PROGRAM sub_Light
VAR
		fbLichtHausgang 		: FB_Light;
		fbLichtTechnikraum 		: FB_Light;
		fbLichtHobbyraum 		: FB_Light;
		fbLichtKueche			: FB_Light;
		fbLichtWerkstatt		: FB_Light;
		fbLichtGarage			: FB_Light;
		fbLichtEsstisch			: FB_LIghtDimm;
		fbLichtBalkon			: FB_LIghtDimm;
		fbLichtEsszimmer		: FB_LightDimmIndirectNC;
		fbLichtWohnzimmer		: FB_LightDimmIndirectNC;
		fbLichtAussenOST		: FB_LightPIR;
		fbLichtAussenHaustur	: FB_LightPIR;
		fbLichtAussenTreppeSud	: FB_LightPIR;
		fbLichtAussenEingang	: FB_LightPIR;
END_VAR

//###################################################################################
//##-----------------------------------BELEUCHTUNG---------------------------------##
//###################################################################################

//--------------------HAUSGANG EG----------------------------------
fbLichtHausgang.bInputs[0] 	:= gvl_EA.bID02_4;
fbLichtHausgang.bInputs[1] 	:= gvl_EA.bID03_1;
fbLichtHausgang.bInputs[2] 	:= gvl_EA.bID03_2;
fbLichtHausgang.bInputs[3] 	:= gvl_EA.bID02_3;

fbLichtHausgang
(
	bInputSec		:= gvl_mb.Output_Coils[242],
	bInputHA		:= gvl_mb.Output_Coils[1],
	bOut 			=> gvl_EA.bOD01_5,
);
//-----------------------------------------------------------------

//--------------------KÜCHE----------------------------------------
fbLichtKueche.bInputs[0]	:= gvl_EA.bID01_4;

fbLichtKueche
(
	bInputSec	:= 	gvl_mb.Output_Coils[242],
	bInputHA	:=	gvl_mb.Output_Coils[0],
	bOut		=>	gvl_EA.bOD01_4, //Licht Küche
	bOut		=>	gvl_EA.bOD04_1,	//Spot Küche
);
//-----------------------------------------------------------------

//--------------------TECHNIKRAUM----------------------------------
fbLichtTechnikraum.bInputs[0] := gvl_EA.bID03_3;

fbLichtTechnikraum
(	
	bInputSec		:= gvl_mb.Output_Coils[242],
	bLightInv_NC	:= TRUE,
	bInputHA		:= gvl_mb.Output_Coils[4],
	bAllFlanks 		:= TRUE,
	bOut 			=> gvl_EA.bOD03_5,
);
//-----------------------------------------------------------------

//--------------------HOBBYRAUM------------------------------------
fbLichtHobbyraum.bInputs[0] := gvl_EA.bID04_1;

fbLichtHobbyraum
(	
	bInputSec		:= gvl_mb.Output_Coils[242],
	bInputHA		:= gvl_mb.Output_Coils[5],
	bAllFlanks 		:= TRUE,
	bOut 			=> gvl_EA.bOD03_1,
	bOut			=> gvl_EA.bOD03_2,
);
//-----------------------------------------------------------------

//--------------------WERKSTATT----------------------------------
fbLichtWerkstatt.bInputs[0] := gvl_EA.bWID01_1;

fbLichtWerkstatt
(	
	bInputSec		:= gvl_mb.Output_Coils[242],
	bLightInv_NC	:= TRUE,
	bInputHA		:= gvl_mb.Output_Coils[6],
	bOut 			=> gvl_EA.bWOD01_1,
);
//-----------------------------------------------------------------

//--------------------GARAGE----------------------------------
fbLichtGarage.bInputs[0] := gvl_EA.bWID01_5;
fbLichtGarage.bInputs[1] := gvl_EA.bWID01_6;

fbLichtGarage
(	
	bInputSec		:= gvl_mb.Output_Coils[242],
	bInputHA		:= gvl_mb.Output_Coils[30],
	bOut 			=> gvl_EA.bWOD01_7,
);
//-----------------------------------------------------------------

//--------------------AUSSEN OST----------------------------------
fbLichtAussenOST
(	
	bInputSecLoop	:= gvl_mb.Output_Coils[243],
	bInputHA		:= gvl_mb.Output_Coils[2],
	bOut 			=> gvl_EA.bOD01_6,
);
//-----------------------------------------------------------------

//--------------------ESSTISCH----------------------------------
fbLichtEsstisch.bInputs[0] := gvl_EA.bID01_3;

fbLichtEsstisch
(	
	bInputSec		:= gvl_mb.Output_Coils[242],
	bInputSecTest	:= gvl_mb.Output_Coils[251],
	bInputHA		:= gvl_mb.Output_Coils[7],
	iDimmValue		:= gvl_mb.Output_Registers[7],
	iNumPress4Dimm	:= 4,
	iOut 			=> gvl_EA.iOADim01,
);
//-----------------------------------------------------------------

//--------------------BALKON----------------------------------
fbLichtBalkon.bInputs[0] := gvl_EA.bID02_2;

fbLichtBalkon
(	
	bInputSec		:= gvl_mb.Output_Coils[243],
	bInputSecTest	:= gvl_mb.Output_Coils[254],
	bInputHA		:= gvl_mb.Output_Coils[10],
	iDimmValue		:= gvl_mb.Output_Registers[10],
	bOnlyAtNight	:= TRUE,
	iNumPress4Dimm	:= 4,
	iOut 			=> gvl_EA.iOADim02,
);
//-----------------------------------------------------------------

//--------------------INDIREKTE BELEUCHTUNG ESSZIMMER--------------
fbLichtEsszimmer.bInputs[0] 	:= gvl_EA.bID01_1;
fbLichtEsszimmer.bInputs[1] 	:= gvl_EA.bID02_1;

fbLichtEsszimmer
(
	bInputSec		:= gvl_mb.Output_Coils[242],
	bInputSecTest	:= gvl_mb.Output_Coils[252],
	bInputHA		:= gvl_mb.Output_Coils[8],
	iDimmValue		:= gvl_mb.Output_Registers[8],
	iNumPress4Dimm	:= 4,
	iOut 			=> gvl_EA.iOA01_2,
	bOut			=> gvl_EA.bOD01_2,
);
//-----------------------------------------------------------------

//--------------------INDIREKTE BELEUCHTUNG WOHNZIMMER-------------
fbLichtWohnzimmer.bInputs[0] 	:= gvl_EA.bID01_2;

fbLichtWohnzimmer
(
	bInputSec		:= gvl_mb.Output_Coils[242],
	bInputSecTest	:= gvl_mb.Output_Coils[253],
	bInputHA		:= gvl_mb.Output_Coils[9],
	iDimmValue		:= gvl_mb.Output_Registers[9],
	iNumPress4Dimm	:= 4,
	iOut 			=> gvl_EA.iOA01_1,
	bOut			=> gvl_EA.bOD01_3,
);
//-----------------------------------------------------------------

//--------------------Aussenbeleuchtung Treppe Süd-------------
fbLichtAussenTreppeSud
(
	bInputSecLoop	:= gvl_mb.Output_Coils[243],
	bInputPIR		:= gvl_ea.bID03_4,
	bInputHA		:= gvl_mb.Output_Coils[28],
	tHigh			:= T#1M,
	bOut			=> gvl_ea.bOD01_8,
);

// Sync PIR to HA
gvl_mb.Output_Coils[29] := gvl_ea.bID03_4;
//-----------------------------------------------------------------

//--------------------Aussenbeleuchtung Eingang Haus-----------
fbLichtAussenEingang
(
	bInputSecLoop	:= gvl_mb.Output_Coils[243],
	bInputPIR		:= gvl_ea.bWID01_7,
	bInputHA		:= gvl_mb.Output_Coils[32],
	tHigh			:= T#1M,
	bOut			=> gvl_ea.bWOD01_8,
);

// Sync PIR to HA
gvl_mb.Output_Coils[31] := gvl_ea.bWID01_7;
//----------------------------------------------------------------

//--------------------AUSSEN HAUSTÜR----------------------------------
fbLichtAussenHaustur
(	
	bInputSecLoop	:= gvl_mb.Output_Coils[243],
	bInputPIR		:= gvl_ea.bWID01_7,
	tHigh			:= T#1M,
	bInputHA		:= gvl_mb.Output_Coils[3],
	bOut 			=> gvl_EA.bOD01_7,
);
//-----------------------------------------------------------------

END_PROGRAM

(* stored: Version 1.1.0.1, ProductVersion 3.1.4024.4
   POU sub_Light: Id {58c72172-b513-4044-8107-df9cb8dc3624}, SpecialFunc None *)
